PROGRAM Move_Axis_Absolute
VAR
	fbMoveAbsolute: MC_MoveAbsolute;
	MoveAbsoluteExecute: BOOL;
	Position: LREAL := 1000;
	Done: BOOL;
END_VAR

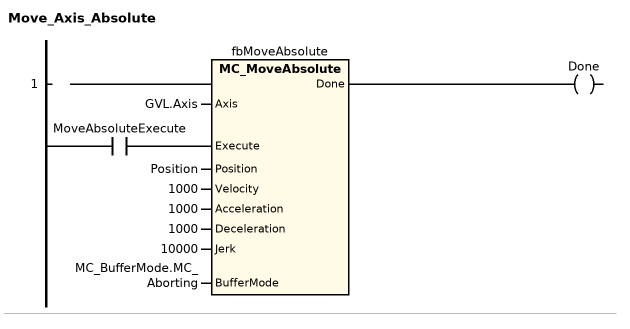
// NETWORK 1
fbMoveAbsolute(
    Axis := GVL.Axis,
    Execute := MoveAbsoluteExecute,
    Position := Position,
    Velocity := 1000,
    Acceleration := 1000,
    Deceleration := 1000,
    Jerk := 10000,
    BufferMode := MC_BufferMode.MC_Aborting); // MC_MoveAbsolute
Done := fbMoveAbsolute.Done;

END_PROGRAM

(* stored: Version 1.1.0.1, ProductVersion 3.1.4024.12
   POU Move_Axis_Absolute: Id {1307d2be-0434-4610-9d94-eeeaf9473cd5}, SpecialFunc None *)
